VAR_GLOBAL
	// Eventlog
	fbEventLog						: FB_Eventlog;	

	// System
	fbSafety						: FB_Safety;
	fbEtherCATBus					: FB_EtherCATBus;
	fbSupervision					: FB_Supervision;	
	
	// Hardware
	fbSafetyLock					: FB_SafetyLock;
	fbMat							: FB_Mat;
	fbPunchEngine					: FB_PunchEngine;
	fbMatAndToolHandling			: FB_MatAndToolHandling;
END_VAR

(* stored: Version 1.1.0.1, ProductVersion 3.1.4022.12
   GVL GVL: Id {ce4e0b60-b7a8-421a-a8f0-c5f124604bf1} *)
